# EPICS substitutions: HeaterIoc/exampleApp/Db/user.substitutions
# Example substitutions file

file "db/dbExample1.db" {
    { user = "hanlf" }
}

file db/dbExample2.db {
    pattern { user, no, scan }
        { "hanlf", 1, "1 second" }
        { "hanlf", 2, "2 second" }
        { "hanlf", 3, "5 second" }
}
